FUNCTION_BLOCK FB_UR5 EXTENDS FB_ROB_MANIP IMPLEMENTS ITF_BA_6Axis, ITF_CommunicationModul
VAR_INPUT
END_VAR
VAR_OUTPUT
END_VAR
VAR
	PiNPl: FB_PickPlaceSkill;
END_VAR

StateMachine();


//Reference to Skills
PiNPl(Rob:=ADR(THIS^));

//ComConfig
ComConfig.sIPAdress:='127.0.0.1';
ComConfig.Port:= 5432;

METHOD M_Connect : BOOL
VAR_INPUT
END_VAR
END_METHOD

METHOD M_Disconnect : BOOL
VAR_INPUT
END_VAR
END_METHOD

METHOD M_ResetConnection : BOOL
VAR_INPUT
END_VAR
END_METHOD

{warning 'Add method implementation '}
METHOD MC_MoveAxesAbsolute : BOOL
VAR_INPUT
	target	: stTarget3D;
END_VAR
IF _state=eState.Active THEN
// 	P_TargetReached:=FALSE;
END_IF
END_METHOD

{warning 'Add method implementation '}
METHOD MC_MoveAxesRelative : BOOL
VAR_INPUT
	axes	: ARRAY [1..6] OF FB_Axis;
	offsets	: ARRAY [1..6] OF REAL;
END_VAR
END_METHOD

{warning 'Add method implementation '}
METHOD MC_MoveLinearAbsolute : BOOL
VAR_INPUT
	target	: stTarget3D;
END_VAR
END_METHOD

{warning 'Add method implementation '}
METHOD MC_ReadActualVelocity : stPose
END_METHOD

{warning 'Add method implementation '}
METHOD MC_ReadAnalogInput : LREAL
VAR_INPUT
	input	: INT;
END_VAR
END_METHOD

{warning 'Add method implementation '}
METHOD MC_ReadDigitalInput : BOOL
VAR_INPUT
	input	: INT;
END_VAR
END_METHOD

{warning 'Add method implementation '}
METHOD MC_SetDigitalOutput : BOOL
VAR_INPUT
	output	: INT;
	value	: BOOL;
END_VAR
END_METHOD

{warning 'Add method implementation '}
METHOD MC_SetOperationMode : BOOL
VAR_INPUT
	mode	: eMode;
END_VAR
_mode:=mode;
END_METHOD

PROPERTY P_bConnected : BOOL
GET
END_GET
END_PROPERTY

END_FUNCTION_BLOCK

(* stored: Version 1.1.0.1, ProductVersion 3.1.4026.18
   POU FB_UR5: Id {7138b06d-6984-4953-8124-68042278758b}, SpecialFunc None
   Folder Communication: Id {962090cd-82cb-4129-9347-c8ac07fb90f4}
   Folder MotionControl: Id {9ed28985-c54d-42fa-8d69-76777d28de96}
   Method M_Connect: Id {ea0b7a54-6a8f-44d8-8b6a-a3c96ae90503}
   Method M_Disconnect: Id {81d53a8c-a37e-4c7e-ab45-5d8abfba1924}
   Method M_ResetConnection: Id {ab760c43-0912-46a9-8200-3ef0d14f05e9}
   Method MC_MoveAxesAbsolute: Id {e4cbbe25-0003-4a3a-941f-ba8ea400b2d6}
   Method MC_MoveAxesRelative: Id {dc6eaf0b-bda4-4a71-9f22-4f43caa591cf}
   Method MC_MoveLinearAbsolute: Id {fac605cc-f9e9-41e9-8d84-7a37c1c2f07e}
   Method MC_ReadActualVelocity: Id {8fcd44ac-c416-4fa2-be4a-a96c08398ed8}
   Method MC_ReadAnalogInput: Id {f3e9cd2c-1bdb-4b96-8862-1b49b481f6f5}
   Method MC_ReadDigitalInput: Id {fa482187-c1ce-433f-9f9a-2cc320aaca90}
   Method MC_SetDigitalOutput: Id {9228931f-d00e-488b-96fa-facc797720c5}
   Method MC_SetOperationMode: Id {b77d92d3-2c73-432f-b915-482766ea505a}
   Property P_bConnected: Id {37ba7a67-b4ee-42b5-aea8-1f3fba5d5175}
   Get Get: Id {d4b74009-4a4c-4abb-b825-78ae2fd94b8a} *)
